(*
## Short summary

This command can be used to create and store a new measurement data set.

.. <legal notes>

legal notes
=================
| SPDX-FileCopyrightText: © 2025 ekvip automation GmbH <info@ekvip.de>
| SPDX-License-Identifier: Apache-2.0
| For details check: Apache-2.0_

.. _Apache-2.0: https://www.apache.org/licenses/LICENSE-2.0

.. </legal notes>

*)
FUNCTION_BLOCK MeasurementAddEntryCommand EXTENDS CNM_AbstractObject.Object IMPLEMENTS CNM_CommandInterfaces.ISingleAttempt
VAR
	recorder :CNM_ProductionMetricInterfaces.IMeasurementRecorder;
	(* product identifier for that specific part *)
	partIdentifier	:Tc2_System.T_MaxString;
	(* name of the measurement, e.g. label position, cell voltage, oven temperature *)
	nameMeasurement	: Tc2_System.T_MaxString;
	(* unit of the measurement, e.g. mm, V, °C *)
	unit	: CNM_ProductionMetricInterfaces.UnitString;
	(* Permissible value range of the measurement for OK parts*)
	range	: CNM_ProductionMetricInterfaces.MeasurementRangeStruct;
	(* value of the measurement *)
	value	: LREAL;
END_VAR

(*

## Short summary

This abstract property returns the class name of the concrete object, 
which is useful for logging/debugging purpose or to check the class name
for ``__DELETE`` in factories (sometimes it's necessary to do more 
than just to free the memory).

.. <legal notes>

legal notes
=================
| SPDX-FileCopyrightText: © 2022 ekvip automation GmbH <info@ekvip.de>
| SPDX-License-Identifier: Apache-2.0
| For details check: Apache-2.0_

.. _Apache-2.0: https://www.apache.org/licenses/LICENSE-2.0

.. </legal notes>

*)
PROPERTY className : CNM_AbstractObject.ClassName
GET
className := 'CNM_ProductionMetrics.CycleTimeStartCycleCommand';
END_GET
END_PROPERTY

(*

## Short summary

Invokes the action associated with this interface.

.. <legal notes>

legal notes
=================
| SPDX-FileCopyrightText: © 2024 ekvip automation GmbH <info@ekvip.de>
| SPDX-License-Identifier: Apache-2.0
| For details check: Apache-2.0_

.. _Apache-2.0: https://www.apache.org/licenses/LICENSE-2.0

.. </legal notes>



*)
METHOD invoke : CNM_ReturnTypes.SingleExecutionResult
IF THIS^.isObjectValid(THIS^.recorder) THEN
	invoke := THIS^.recorder.addMeasurementEntry(
		partIdentifier := THIS^.partIdentifier,
		name := THIS^.nameMeasurement,
		unit := THIS^.unit,
		range := THIS^.range,
		value := THIS^.value
	);
ELSE
	invoke := CNM_ReturnTypes.SingleExecutionResult.ABORTED;
END_IF
END_METHOD

METHOD INTERNAL setParameters
VAR_INPUT
	(* product identifier for that specific part *)
	partIdentifier	:Tc2_System.T_MaxString;
	(* name of the measurement, e.g. label position, cell voltage, oven temperature *)
	name	: Tc2_System.T_MaxString;
	(* unit of the measurement, e.g. mm, V, °C *)
	unit	: CNM_ProductionMetricInterfaces.UnitString;
	(* Permissible value range of the measurement for OK parts*)
	range	: CNM_ProductionMetricInterfaces.MeasurementRangeStruct;
	(* value of the measurement *)
	value	: LREAL;
END_VAR
THIS^.partIdentifier := partIdentifier;
THIS^.nameMeasurement := name;
THIS^.unit := unit;
THIS^.range := range;
THIS^.value := value;
END_METHOD

(*
## Short summary

This methods sets the cycletime recorder interface on which the command is executed.

.. <legal notes>

legal notes
=================
| SPDX-FileCopyrightText: © 2025 ekvip automation GmbH <info@ekvip.de>
| SPDX-License-Identifier: Apache-2.0
| For details check: Apache-2.0_

.. _Apache-2.0: https://www.apache.org/licenses/LICENSE-2.0

.. </legal notes>

*)

METHOD setRecorder
VAR_INPUT
	recorder :CNM_ProductionMetricInterfaces.IMeasurementRecorder;
END_VAR
IF THIS^.isObjectValid(recorder) THEN
	THIS^.recorder := recorder;
END_IF
END_METHOD

END_FUNCTION_BLOCK

(* stored: Version 1.1.0.1
   POU MeasurementAddEntryCommand: Id {144f2467-47e7-4325-b6ee-6ff4b8b2d3f7}, SpecialFunc None
   Property className: Id {fdb0f910-57be-4107-aad2-e2b6a78c1e0d}
   Get Get: Id {f33d5b17-2b48-4477-b5d1-cc7aadc99025}
   Method invoke: Id {92a344b2-dd6c-4b47-addb-626601c1a88e}
   Method setParameters: Id {d2bb7239-ebdd-492d-b25f-48e8c5b01a0d}
   Method setRecorder: Id {51c675e0-2f63-406d-a0e9-4a5575d504a9} *)
